(* Logix 5000 project; controller traffic_light 1769-L16ER-BB1B rev 32.11; software revision 32.00 *)

TASK MainTask (continuous, watchdog 500 ms) : MainProgram

MODULES
   Local : 1769-L16ER-BB1B (PointIO 0, rev 32.11)
      Discrete_IO : Embedded (PointIO 1, rev 32.11, Output RPI 20 ms)
END_MODULES

PROGRAM MainProgram   (* main routine MainRoutine *)
VAR
   b0 : BOOL;
   b1 : BOOL;
   b2 : BOOL;
   b3 : BOOL;
   b4 : BOOL;
   Green_EW : BOOL;
   Green_NS : BOOL;
   Green_NS_Turn : BOOL;
   Red_EW : BOOL;
   Red_NS : BOOL := 1;
   Red_NS_Turn : BOOL := 1;
   timer1 : TIMER := (PRE := 3, ACC := 3, EN := 1, DN := 1);
   timer2 : TIMER := (PRE := 3, ACC := 3, EN := 1, DN := 1);
   timer3 : TIMER := (PRE := 3, ACC := 3, EN := 1, DN := 1);
   timer4 : TIMER := (PRE := 3, ACC := 3, EN := 1, DN := 1);
   timer5 : TIMER := (PRE := 3, EN := 1, TT := 1);
   timer6 : TIMER := (PRE := 3);
   Yellow_EW : BOOL := 1;
   Yellow_NS : BOOL;
   Yellow_NS_Turn : BOOL;
END_VAR

ROUTINE MainRoutine   (* ladder *)
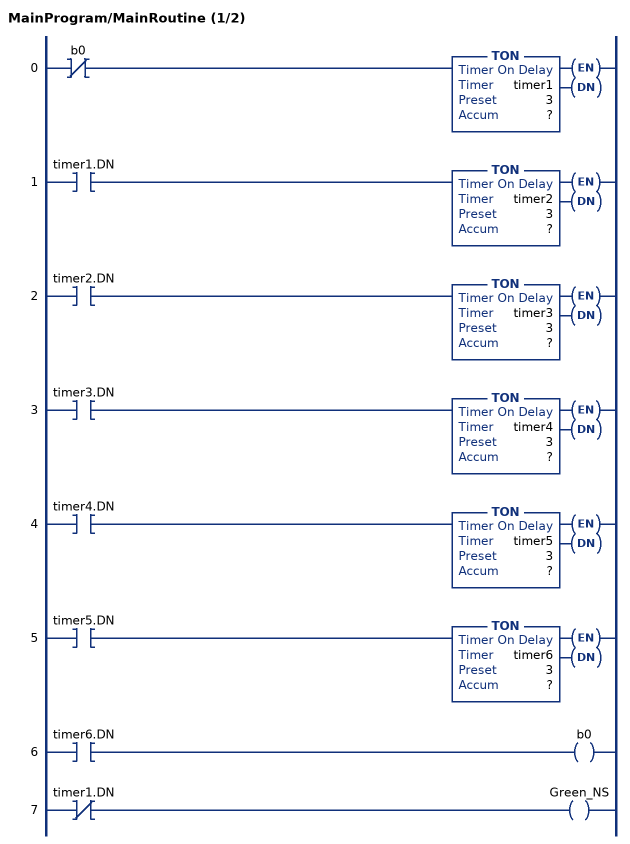
   0: XIO(b0)TON(timer1,?,?);
   1: XIC(timer1.DN)TON(timer2,?,?);
   2: XIC(timer2.DN)TON(timer3,?,?);
   3: XIC(timer3.DN)TON(timer4,?,?);
   4: XIC(timer4.DN)TON(timer5,?,?);
   5: XIC(timer5.DN)TON(timer6,?,?);
   6: XIC(timer6.DN)OTE(b0);
   7: XIO(timer1.DN)OTE(Green_NS);
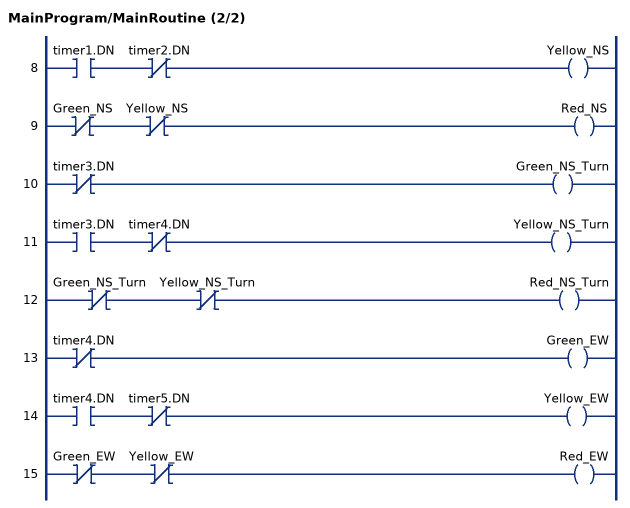
   8: XIC(timer1.DN)XIO(timer2.DN)OTE(Yellow_NS);
   9: XIO(Green_NS)XIO(Yellow_NS)OTE(Red_NS);
   10: XIO(timer3.DN)OTE(Green_NS_Turn);
   11: XIC(timer3.DN)XIO(timer4.DN)OTE(Yellow_NS_Turn);
   12: XIO(Green_NS_Turn)XIO(Yellow_NS_Turn)OTE(Red_NS_Turn);
   13: XIO(timer4.DN)OTE(Green_EW);
   14: XIC(timer4.DN)XIO(timer5.DN)OTE(Yellow_EW);
   15: XIO(Green_EW)XIO(Yellow_EW)OTE(Red_EW);
END_ROUTINE
END_PROGRAM
